// This function Block extends the Referenced Library Mover (FB), so the user can expand the capabilities of the XTS Mover Functions
FUNCTION_BLOCK ApplicationMover EXTENDS Mover
VAR_INPUT
END_VAR
VAR_OUTPUT
END_VAR
VAR
	_PositionLag: LREAL;

END_VAR

METHOD Cyclic : iMover
VAR_IN_OUT
	GroupReference	: AXES_GROUP_REF;
END_VAR
// Call Base Class (Mover) Cyclic Logic
SUPER^.Cyclic(GroupReference);

//======= 
// To Call ApplicationMover addon Method/Properties/Variables... 
//		you must call Mover[] array index directly, as Station/Zone/PositionTrig/SpeedTrig do not know about ApplicationMover add ons

// Add ApplicationMover specific code here

// example position lag property
_PositionLag:= THIS^.AxisReference.NcToPlc.PosDiff;

// Latch Errors

// Call Fbs Cyclically
END_METHOD

{attribute 'monitoring' := 'call'}
PROPERTY PositionLag : LREAL
GET
PositionLag:= _PositionLag;
END_GET
END_PROPERTY

END_FUNCTION_BLOCK

(* stored: Version 1.1.0.1, ProductVersion 3.1.4026.18
   POU ApplicationMover: Id {516536b5-5233-0a95-01e8-9585147c75fa}, SpecialFunc None
   Method Cyclic: Id {a81886a0-983c-0294-0adc-9591fa48a449}
   Property PositionLag: Id {2f9b4da0-9f46-0501-2862-3b56ba7816bb}
   Get Get: Id {8ea91099-3f22-02ba-0930-a3b600f2f5d6} *)
